// TIA Portal V18 export
DATA_BLOCK "Multi instance FB_DB"   // DB4
VERSION : 0.1
// stored: AutoNumber true, DBAccessibleFromOPCUA true, InstanceOfName Multi instance FB, InstanceOfType FB
"Multi instance FB"
   // VAR
   //    "Motor control function FB_Instance" { S7_SetPoint := 'True'} : "Motor control function FB";
   //    "Motor control function FB_Instance_1" { S7_SetPoint := 'True'} : "Motor control function FB";
   // END_VAR
BEGIN
END_DATA_BLOCK
